Universal Robots PolyScope program: shaft_centering_in_vgroove.urp

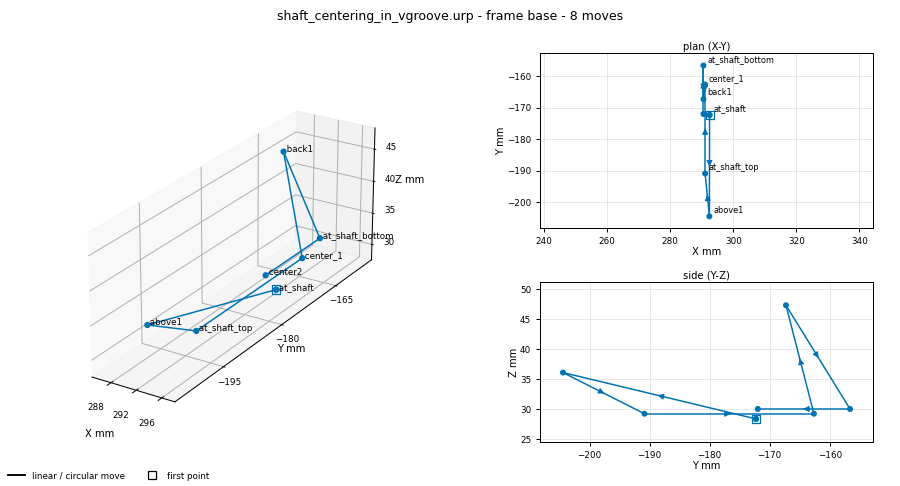
[picture p0: tool path of shaft_centering_in_vgroove.urp in frame base, 8 of 9 moves have a stored position in this frame; points joined in program order, loops and branches not executed]
Program shaft_centering_in_vgroove (installation=default directory=/programs/wrs2020 createdIn=5.7.0.90932 lastSavedIn=5.10.0.106288 robotSerialNumber=20205500607)
Calibrated DH parameters: a=[0.000096, -0.337, -0.383372, 0.000118, 0.000015, 0]; d=[0.162724, 79.377998, -95.545185, 16.300583, 0.099689, 0.099499]; alpha=[1.569249, 0.003272, 0.005201, 1.570041, -1.570219, 0]; deltaTheta=[0, 0.65664, 5.410619, 0.215927, -0.000001, 0]
Robot Program (runOnlyOnce=false)
  URCap Gripper (Robotiq_Grippers, Robotiq Inc.) dataModel(position=0.0, force=100.0, speed=100.0, positionInDouble=0.0, forceInDouble=100.0, speedInDouble=100.0, slaveIds=[9], blocking=true)
  MoveL speed 800 mm/s, acceleration 1200 mm/s^2 (useActiveTCP=true) feature=Base
    Waypoint at_shaft: motionParameters(blendRadius=0.01); TCP in base x=292.462 y=-172.285 z=28.427 mm, rx=-0.0168 ry=3.1097 rz=0.0286 rad; joints [124.781, -97.407, 145.354, -138.076, -87.656, 34.218] deg; TCP offset x=0 y=0 z=165 mm, rx=0 ry=0 rz=0 rad
    Waypoint above1: motionParameters(blendRadius=0.007); TCP in base x=292.406 y=-204.446 z=36.152 mm, rx=-1.067 ry=2.8561 rz=0.2258 rad; joints [118.482, -93.042, 137.84, -127.028, -83.785, -12.882] deg
    Waypoint at_shaft_top: motionParameters(blendRadius=0.005); TCP in base x=291.051 y=-190.872 z=29.293 mm, rx=-2.0595 ry=2.0908 rz=0.2351 rad; joints [117.619, -91.659, 137.377, -123.568, -81.624, -62.386] deg
    Waypoint center_1: motionParameters(jointSpeed=1.047198 jointAcceleration=1.396263 cartesianSpeed=0.25 cartesianAcceleration=1.2); TCP in base x=291.051 y=-162.634 z=29.293 mm, rx=-2.0595 ry=2.0908 rz=0.2351 rad; joints [119.845, -94.395, 140.006, -123.779, -81.171, -60.188] deg
  MoveL speed 800 mm/s, acceleration 1200 mm/s^2 (useActiveTCP=true) feature=Base
    Waypoint back1: motionParameters(blendRadius=0.01); TCP in base x=290.517 y=-167.295 z=47.369 mm, rx=-2.1574 ry=2.1953 rz=0.0422 rad; joints [124.002, -100.498, 143.014, -130.277, -86.462, -55.049] deg
    Waypoint at_shaft_bottom: motionParameters(blendRadius=0.005); TCP in base x=290.517 y=-156.619 z=30.083 mm, rx=2.104 ry=-2.1459 rz=0.242 rad; joints [134.153, -99.166, 151.109, -151.176, -96.961, -45.193] deg
    Waypoint center2: motionParameters(jointSpeed=1.047198 jointAcceleration=1.396263 cartesianSpeed=0.25 cartesianAcceleration=1.2); TCP in base x=290.517 y=-171.985 z=30.083 mm, rx=2.104 ry=-2.1459 rz=0.242 rad; joints [131.971, -98.009, 150.364, -151.853, -96.603, -47.357] deg
    Waypoint back2 (Relative): motionParameters(blendRadius=0.004); relativeFromPosition TCP in base x=290.486 y=-171.972 z=30.053 mm, rx=2.104 ry=-2.1459 rz=0.2418 rad; joints [131.969, -98.008, 150.367, -151.853, -96.603, -47.357] deg; TCP in base x=290.523 y=-163.583 z=30.089 mm, rx=2.1041 ry=-2.1459 rz=0.242 rad; joints [133.148, -98.652, 150.784, -151.49, -96.796, -46.191] deg
    Waypoint at_shaft: TCP in base x=292.462 y=-172.285 z=28.427 mm, rx=-0.0168 ry=3.1097 rz=0.0286 rad; joints [124.781, -97.407, 145.354, -138.076, -87.656, 34.218] deg
